(* PLC project ProgramaTCC.project, MasterTool IEC XE MasterTool IEC XE *)
(* stored: creationDateTime 2021-03-26T21:36:05.1270446, modificationDateTime 2021-03-26T21:29:27.7889283 *)

(* Main POU associated with MainTask that calls StartPrg, UserPrg/ActivePrg and NonSkippedPrg. This POU is blocked to edit. *)
PROGRAM MainPrg
  VAR
    isFirstCycle : BOOL := TRUE;
  END_VAR

                    SpecialVariablesPrg();
IF isFirstCycle THEN
   StartPrg();
   isFirstCycle := FALSE;
ELSE
   UserPrg();
END_IF;
                  
END_PROGRAM

(* The main code inserted by the user and executed associated with the MainTask must be inserted into this POU. *)
PROGRAM UserPrg
  VAR
    Botao1 : BOOL;
    Lampada1 : BOOL;
    TON_1 : TON;
    Lampada2 : BOOL;
  END_VAR

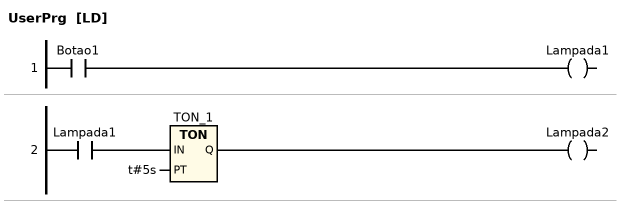
(* LD diagram, written out as Structured Text *)
(* Ao Acionar o Botao1, a Lampada1 irá acender *)

Lampada1 := Botao1;
(* Após acender a Lampada1 irá iniciar uma contagem de 5 segundo e após terminar a contagem, a Lampada2 irá acender *)

TON_1(IN := Lampada1, PT := t#5s);
Lampada2 := TON_1.Q;
END_PROGRAM

(* The code inserted by the user into this POU is executed once after startup. Before this fist cycle it is not executed again. In case of redundant system, this one is executed in both CPUs during the startup. *)
PROGRAM StartPrg

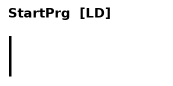
(* LD diagram, written out as Structured Text *)
(* --- network --- *)
END_PROGRAM

(* This POU is blocked to edit. *)
{attribute 'hide'}
PROGRAM SpecialVariablesPrg
  VAR
    udiMicroAcc : UDINT;  (* Microseconds accumulator *)
  END_VAR

                    // Update pulse bits
udiMicroAcc:= udiMicroAcc + Special_Variables.udiMainTaskInterval;
IF udiMicroAcc MOD 100000 >= 50000 THEN Pulse_100ms:= TRUE; ELSE Pulse_100ms:= FALSE; END_IF
IF udiMicroAcc MOD 500000 >= 250000 THEN Pulse_500ms:= TRUE; ELSE Pulse_500ms:= FALSE; END_IF
IF udiMicroAcc MOD 1000000 >= 500000 THEN Pulse_1s:= TRUE; ELSE Pulse_1s:= FALSE; END_IF
IF udiMicroAcc MOD 2000000 >= 1000000 THEN Pulse_2s:= TRUE; ELSE Pulse_2s:= FALSE; END_IF
IF udiMicroAcc MOD 5000000 >= 2500000 THEN Pulse_5s:= TRUE; ELSE Pulse_5s:= FALSE; END_IF
IF udiMicroAcc MOD 10000000 >= 5000000 THEN Pulse_10s:= TRUE; ELSE Pulse_10s:= FALSE; END_IF
IF udiMicroAcc MOD 30000000 >= 15000000 THEN Pulse_30s:= TRUE; ELSE Pulse_30s:= FALSE; END_IF
IF udiMicroAcc MOD 60000000 >= 30000000 THEN Pulse_60s:= TRUE; ELSE Pulse_60s:= FALSE; END_IF
udiMicroAcc:= udiMicroAcc MOD 120000000;

// Update scan pulse
Pulse_Scan:= NOT Pulse_Scan;

// Update system time
GetDateAndTime(System_Time);

// Update Hour_Minute
Hour_Minute:= System_Time.byHours * 100 + System_Time.byMinutes;

// Update Day of Week
Day_Of_Week:= GetDayOfWeek();
                  
END_PROGRAM

CONFIGURATION Device
  RESOURCE Application ON PLC
    VAR_GLOBAL  (* System_Diagnostics *)
      DG_NX3003 AT %QB21040 : T_DIAG_NX3003_1;  (* DG_NX3003 diagnostics variable *)
    END_VAR
    VAR_GLOBAL  (* Special_Variables - This GVL is blocked to edit. *)
      Pulse_100ms : BOOL;  (* Pulse signal with 100ms period (toggles every 50ms) *)
      Pulse_500ms : BOOL;  (* Pulse signal with 500ms period (toggles every 250ms) *)
      Pulse_1s : BOOL;  (* Pulse signal with 1s period (toggles every 500ms) *)
      Pulse_2s : BOOL;  (* Pulse signal with 2s period (toggles every 1s) *)
      Pulse_5s : BOOL;  (* Pulse signal with 5s period (toggles every 2,5s) *)
      Pulse_10s : BOOL;  (* Pulse signal with 10s period (toggles every 5s) *)
      Pulse_30s : BOOL;  (* Pulse signal with 30s period (toggles every 15s) *)
      Pulse_60s : BOOL;  (* Pulse signal with 60s period (toggles every 30s) *)
      Pulse_Scan : BOOL;  (* Scan pulse that toggles every MainTask cycle *)
      System_Time : EXTENDED_DATE_AND_TIME;  (* System date and time *)
      Day_Of_Week : DAYS_OF_WEEK;  (* Day of week *)
      Hour_Minute : UINT;  (* Integer variable with hour and minute (hour*100 + minute) *)
      udiMainTaskInterval : UDINT := 20000;  (* MainTask configured interval [us]. *)
    END_VAR
    VAR_GLOBAL  (* IntegratedIO *)
      DigitalInputs : T_DIGITAL_INPUTS_2;  (* Digital Inputs structure *)
      DigitalOutputs : T_DIGITAL_OUTPUTS_2;  (* Digital Outputs structure *)
      FastInputs : T_FAST_INPUTS_2;  (* Fast Inputs structure *)
      FastOutputs : T_FAST_OUTPUTS_2;  (* Fast Outputs structure *)
      I00 : REFERENCE TO BOOL := DigitalInputs.I00;  (* Digital Input 00 *)
      I01 : REFERENCE TO BOOL := DigitalInputs.I01;  (* Digital Input 01 *)
      I02 : REFERENCE TO BOOL := DigitalInputs.I02;  (* Digital Input 02 *)
      I03 : REFERENCE TO BOOL := DigitalInputs.I03;  (* Digital Input 03 *)
      I04 : REFERENCE TO BOOL := DigitalInputs.I04;  (* Digital Input 04 *)
      I05 : REFERENCE TO BOOL := DigitalInputs.I05;  (* Digital Input 05 *)
      I06 : REFERENCE TO BOOL := DigitalInputs.I06;  (* Digital Input 06 *)
      I07 : REFERENCE TO BOOL := DigitalInputs.I07;  (* Digital Input 07 *)
      I08 : REFERENCE TO BOOL := DigitalInputs.I08;  (* Digital Input 08 *)
      I09 : REFERENCE TO BOOL := DigitalInputs.I09;  (* Digital Input 09 *)
      I10 : REFERENCE TO BOOL := DigitalInputs.I10;  (* Digital Input 10 *)
      I11 : REFERENCE TO BOOL := DigitalInputs.I11;  (* Digital Input 11 *)
      I12 : REFERENCE TO BOOL := DigitalInputs.I12;  (* Digital Input 12 *)
      I13 : REFERENCE TO BOOL := DigitalInputs.I13;  (* Digital Input 13 *)
      Q00 : REFERENCE TO BOOL := DigitalOutputs.Q00;  (* Digital Output 00 *)
      Q01 : REFERENCE TO BOOL := DigitalOutputs.Q01;  (* Digital Output 01 *)
      Q02 : REFERENCE TO BOOL := DigitalOutputs.Q02;  (* Digital Output 02 *)
      Q03 : REFERENCE TO BOOL := DigitalOutputs.Q03;  (* Digital Output 03 *)
      Q04 : REFERENCE TO BOOL := DigitalOutputs.Q04;  (* Digital Output 04 *)
      Q05 : REFERENCE TO BOOL := DigitalOutputs.Q05;  (* Digital Output 05 *)
      Q06 : REFERENCE TO BOOL := DigitalOutputs.Q06;  (* Digital Output 06 *)
      Q07 : REFERENCE TO BOOL := DigitalOutputs.Q07;  (* Digital Output 07 *)
      Q08 : REFERENCE TO BOOL := DigitalOutputs.Q08;  (* Digital Output 08 *)
      Q09 : REFERENCE TO BOOL := DigitalOutputs.Q09;  (* Digital Output 09 *)
    END_VAR
    TASK Configuration(INTERVAL := T#5ms, PRIORITY := 4);
    TASK MainTask(INTERVAL := T#20ms, PRIORITY := 13);
    PROGRAM Configuration.EtherCAT_Task WITH Configuration : Configuration.EtherCAT_Task;
    PROGRAM MainPrg WITH MainTask : MainPrg;
  END_RESOURCE
END_CONFIGURATION

CONFIGURATION Configuration
END_CONFIGURATION

CONFIGURATION NX3003
END_CONFIGURATION

CONFIGURATION <Vazio>
END_CONFIGURATION

CONFIGURATION COM 1
END_CONFIGURATION

CONFIGURATION NET 1
END_CONFIGURATION

CONFIGURATION Integrated I/O
END_CONFIGURATION
